# EPICS autosave request: xspress3App/Db/xsp3.req
file "NDFileHDF5_settings.req", P=$(P), R=HDF1:
